FUNCTION_BLOCK TYPE_DETECTOR (* Basic FB with empty ECC *)
  (* Standard: 61499-2 *)
  (* Version 1.0, 2023-04-20, valentinnodan *)
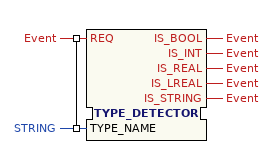
  EVENT_INPUT
    REQ WITH TYPE_NAME;
  END_EVENT
  EVENT_OUTPUT
    IS_BOOL;
    IS_INT;
    IS_REAL;
    IS_LREAL;
    IS_STRING;
  END_EVENT
  VAR_INPUT
    TYPE_NAME : STRING;
  END_VAR
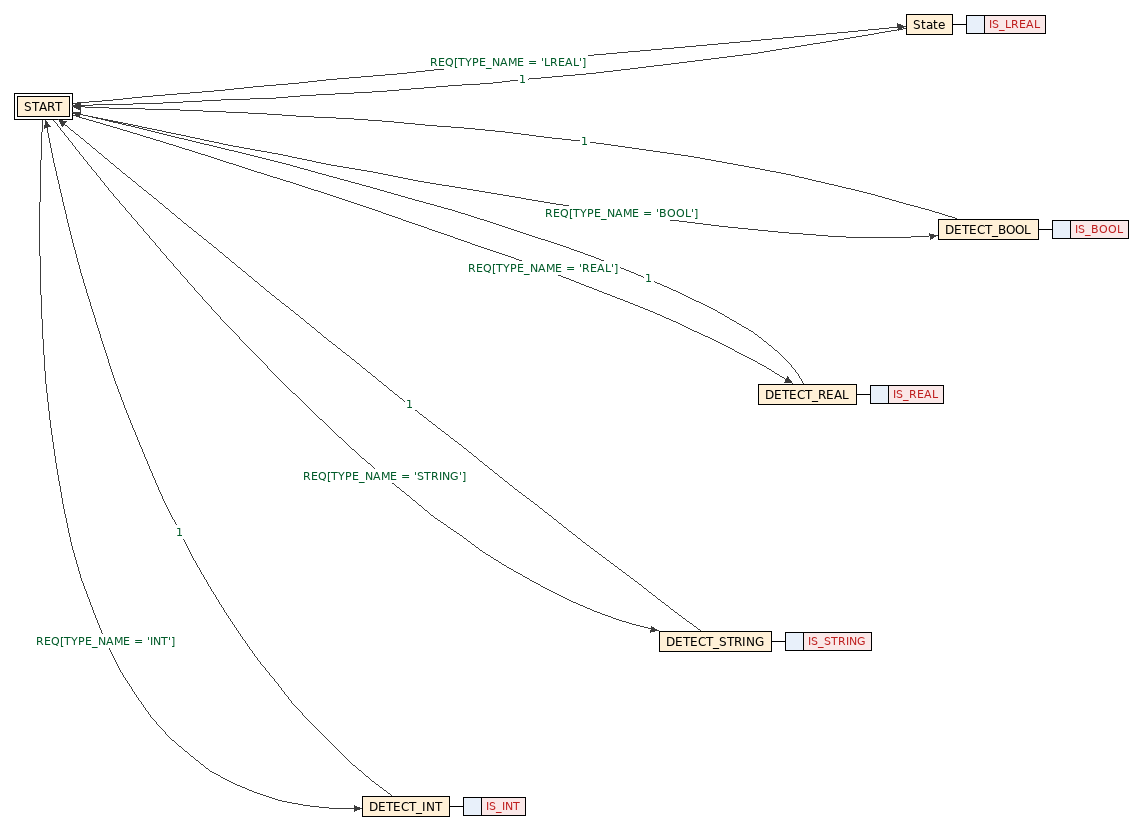
  EC_STATES
    START; (* Initial State *)
    DETECT_BOOL : -> IS_BOOL;
    DETECT_REAL : -> IS_REAL;
    DETECT_STRING : -> IS_STRING;
    DETECT_INT : -> IS_INT;
    State : -> IS_LREAL;
  END_STATES
  EC_TRANSITIONS
    START TO DETECT_BOOL := REQ[TYPE_NAME = 'BOOL'];
    DETECT_BOOL TO START := 1;
    START TO DETECT_REAL := REQ[TYPE_NAME = 'REAL'];
    DETECT_REAL TO START := 1;
    START TO DETECT_STRING := REQ[TYPE_NAME = 'STRING'];
    DETECT_STRING TO START := 1;
    START TO DETECT_INT := REQ[TYPE_NAME = 'INT'];
    DETECT_INT TO START := 1;
    START TO State := REQ[TYPE_NAME = 'LREAL'];
    State TO START := 1;
  END_TRANSITIONS
END_FUNCTION_BLOCK
